(* This function block is created for interface devices between different PLC*)
(* Not all the fields in the original structure is required, just few signals *)
FUNCTION_BLOCK FB_TVCG_ADS
VAR_INPUT
	sNetId : String; //NetID of the Destination PLC controller
	nPort : int; // port number
	sVarName : string;// the variable name of the declared function block.

END_VAR
VAR_OUTPUT
	{attribute 'pytmc' := 'pv: '}
	VGC:ST_VGC;
END_VAR
VAR
	xOpnLS 	: BOOL;
	xClsLS 	: BOOL;
	
	fb_Read_xOpnLS: FB_ReadAdsSymByName;
	fb_Read_xClsLS: FB_ReadAdsSymByName;
	ftReset_xOpnLS: F_TRIG;
	ftReset_xClsLS: F_TRIG;
	xFirstPass: bool:= true;
END_VAR

ftReset_xOpnLS(CLK:= fb_Read_xOpnLS.bBusy OR xFirstPass);
ftReset_xClsLS(CLK:= fb_Read_xClsLS.bBusy OR xFirstPass);
(*calling ADS read function*)
fb_Read_xOpnLS(
	bRead:= ftReset_xOpnLS.Q, 
	sNetId:= sNetId, 
	nPort:= nPort, 
	sVarName:= CONCAT(sVarName,'iq_stValve.i_xOpnLS'), 
	nDestAddr:= ADR(xOpnLS), 
	nLen:= SIZEOF(xOpnLS), 
	tTimeout:= , 
	eComMode:= , 
	bBusy=> , 
	bError=> , 
	nErrorId=> );
	
fb_Read_xClsLS(
	bRead:= ftReset_xClsLS.Q, 
	sNetId:= sNetId, 
	nPort:= nPort, 
	sVarName:= CONCAT(sVarName,'iq_stValve.i_xClsLS'), 
	nDestAddr:= ADR(xClsLS), 
	nLen:= SIZEOF(xClsLS), 
	tTimeout:= , 
	eComMode:= , 
	bBusy=> , 
	bError=> , 
	nErrorId=> );

(*Soft Io mapping*)
VGC.i_xClsLS := xClsLS;
VGC.i_xOpnLS := xOpnLS;

END_FUNCTION_BLOCK

(* stored: Version 1.1.0.1, ProductVersion 3.1.4024.0
   POU FB_TVCG_ADS: Id {84085701-3a86-43d0-96fb-51ae4e0cc36d}, SpecialFunc None *)
